// TwinCAT 3 PLC project TcMotionInterface_Test
// Title: TcMotionInterface_Test
// Company: TcInterfaces
// Author: R&B
// ProjectVersion: 1.0.0.0
// ProgramVersion: 3.1.4026.22
// CompilerDefines: ,VISU_USEPROPERTYINFO
// libraries:
//   Tc2_MC2, * (Beckhoff Automation GmbH)
//   Tc2_System, * (Beckhoff Automation GmbH)
//   Tc2_Utilities, * (Beckhoff Automation GmbH)
//   [TcMotionInterface], * (TcInterfaces)
//   VisuDialogs
// project tree:
//   / GlobalTextList.TcGTLO, PlcTask.TcTTO, PRG_TEST.TcPOU, Visualization Manager.TcVMO (not stored)
//   GVLs/ GVL.TcGVL
//   TESTs/ MotionTest.TcPOU (not stored), NcParameterTest.TcPOU (not stored), View_Test.TcVIS, XmlHandler_Test.TcPOU
// real-time tasks:
//   TASK PlcTask: cycle T#1ms, priority 6, ADS port 350
// motion (NC):
//   TASK NC-Task 1 SAF: cycle T#1ms, priority 4, ADS port 501
//   TASK NC-Task 1 SVB: cycle T#1ms, priority 8, ADS port 511
//   AXIS Axis1 (id 1)
//     MotionControl: Range=1, Time=1
//     OtherSettings: AllowMotionCmdToSlave=true
//     encoder EncType=16
//       EncPara: MaxCount=#x0000ffff
//     drive DrvType=13
//       Analog: TorqueSetpointScale=10, ScaleFactorActTorque=0.1
//       TimeComp: TaskDelayCycles=1
//     controller CtrType=1
//       CtrPara: PriorControlFactor=1
//         Observer: BandWidth=20
//   AXIS Axis2 (id 2)
//     OtherSettings: AllowMotionCmdToSlave=true
//     encoder EncType=16
//       EncPara: MaxCount=#x0000ffff
//     drive DrvType=13
//       Analog: TorqueSetpointScale=10, ScaleFactorActTorque=0.1
//       TimeComp: TaskDelayCycles=1
//     controller CtrType=1
//       CtrPara: PriorControlFactor=1
//         Observer: BandWidth=20
//   AXIS Axis3 (id 3)
//     OtherSettings: AllowMotionCmdToSlave=true
//     encoder EncType=16
//       EncPara: MaxCount=#x0000ffff
//     drive DrvType=13
//       Analog: TorqueSetpointScale=10, ScaleFactorActTorque=0.1
//       TimeComp: TaskDelayCycles=1
//     controller CtrType=1
//       CtrPara: PriorControlFactor=1
//         Observer: BandWidth=20
// variable links:
//   __THIS__ <-> TcMotionInterface_Test/TcMotionInterface_Test Instance
//     Inputs/FromPlc <-> PlcTask Outputs/GVL.axRef[0].PlcToNc
//     Inputs/FromPlc <-> PlcTask Outputs/GVL.axRef[1].PlcToNc
//     Inputs/FromPlc <-> PlcTask Outputs/GVL.axRef[2].PlcToNc
//     Outputs/ToPlc <-> PlcTask Inputs/GVL.axRef[0].NcToPlc
//     Outputs/ToPlc <-> PlcTask Inputs/GVL.axRef[1].NcToPlc
//     Outputs/ToPlc <-> PlcTask Inputs/GVL.axRef[2].NcToPlc
//   __THIS__ <-> MotionControllerLibrary/MotionControllerLibrary Instance
//     Inputs/FromPlc <-> PlcTask Outputs/GVL.axRef[0].PlcToNc
//     Inputs/FromPlc <-> PlcTask Outputs/GVL.axRef[1].PlcToNc
//     Inputs/FromPlc <-> PlcTask Outputs/GVL.axRef[2].PlcToNc
//     Outputs/ToPlc <-> PlcTask Inputs/GVL.axRef[0].NcToPlc
//     Outputs/ToPlc <-> PlcTask Inputs/GVL.axRef[1].NcToPlc
//     Outputs/ToPlc <-> PlcTask Inputs/GVL.axRef[2].NcToPlc
//   (this object) <-> TcMotionInterface_Test/TcMotionInterface_Test Instance
//     Inputs/FromPlc <-> PlcTask Outputs/GVL.axRef[0].PlcToNc
//     Inputs/FromPlc <-> PlcTask Outputs/GVL.axRef[1].PlcToNc
//     Inputs/FromPlc <-> PlcTask Outputs/GVL.axRef[2].PlcToNc
//     Outputs/ToPlc <-> PlcTask Inputs/GVL.axRef[0].NcToPlc
//     Outputs/ToPlc <-> PlcTask Inputs/GVL.axRef[1].NcToPlc
//     Outputs/ToPlc <-> PlcTask Inputs/GVL.axRef[2].NcToPlc

CONFIGURATION TcMotionInterface_Test
    RESOURCE PLC ON TwinCAT3
        TASK PlcTask(INTERVAL := T#1ms, PRIORITY := 6);
        PROGRAM PRG_TEST WITH PlcTask : PRG_TEST;
    END_RESOURCE
END_CONFIGURATION

// ---- GVLs/GVL.TcGVL
{attribute 'qualified_only'}
VAR_GLOBAL
	{attribute 'TcNcAxis' := '[0]:=Axis1; [1]:=Axis2; [2]:= Axis3'}
	axRef: ARRAY[0..2] OF AXIS_REF;
END_VAR

// ---- PRG_TEST.TcPOU
PROGRAM PRG_TEST
VAR
	Motion	: MotionTest;
	NC		: NcParameterTest;
	XML		: XmlHandler_Test;
END_VAR

Motion();
NC();
XML();

END_PROGRAM

// ---- TESTs/XmlHandler_Test.TcPOU
FUNCTION_BLOCK XmlHandler_Test
VAR
	XmlHandler: TcDriveParameterHandler;
	RouterMem: FB_GetRouterStatusInfo;
	Status: ST_TcRouterStatusInfo;
	file: STRING := '/home/Administrator/parm.xml';
	file2: STRING := '/home/Administrator/i550V5_4_Async50HzV1.xml';
	ax: AXIS_REF;
	write: BOOL;
	write2: BOOL;
	powerOn: BOOL;
	readState: BOOL;
	readAddr: BOOL;
	power: MC_Power;
	state: MC_ReadStatus;
	address: MC_ReadDriveAddress;
	reset: BOOL;
	starter: BOOL;
	startTime: ULINT;
	stopTime: ULINT;
	diffTime: ULINT;
	parametersWritten: UDINT;
	parametersWritten2: UDINT;
	canAms: STRING := '192.168.17.10.3.1';
	canNode: UINT := 14;
END_VAR

IF powerOn THEN
	power(Axis:= ax, 
		Enable:= TRUE, 
		Enable_Positive:= TRUE, 
		Enable_Negative:= TRUE
	);
END_IF

IF readState THEN
	state(Axis:= ax, Enable:= TRUE);
END_IF

IF readAddr THEN
	address(Axis:= ax, Execute:= TRUE);
END_IF

IF write and not write2 THEN
	IF NOT starter THEN
		startTime := F_GetSystemTime();
		starter := TRUE;
	END_IF
	
	IF XmlHandler.WriteEtcDriveParameter(FilePath:= file, NetId:= ax.DriveAddress.NetID, EtcAddress:= ax.DriveAddress.SlaveAddress, NumberOfParameterWritten=> parametersWritten) THEN
		stopTime := F_GetSystemTime();
		diffTime := (stopTime - startTime) / 10000; // ms
		starter := FALSE;
		write := FALSE;
	END_IF
	IF XmlHandler.Error THEN
		starter := FALSE;
		write := FALSE;
	END_IF
END_IF

IF write2 AND NOT write THEN
	IF NOT starter THEN
		startTime := F_GetSystemTime();
		starter := TRUE;
	END_IF
	
	IF XmlHandler.WriteCanOpenParameters(FilePath:= file2, NetId:= canAms, CanId:= canNode, NumberOfParameterWritten=> parametersWritten2) THEN
		stopTime := F_GetSystemTime();
		diffTime := (stopTime - startTime) / 10000; // ms
		starter := FALSE;
		write2 := FALSE;
	END_IF
	IF XmlHandler.Error THEN
		starter := FALSE;
		write2 := FALSE;
	END_IF
END_IF

IF reset THEN
	XmlHandler.ResetError();
	reset := FALSE;
END_IF

RouterMem(bExecute:= TRUE);
IF NOT RouterMem.bBusy THEN
	Status := RouterMem.info;
	RouterMem(bExecute:= FALSE);
END_IF

END_FUNCTION_BLOCK

// ---- GlobalTextList.TcGTLO
TEXTLIST GlobalTextList
  181 = '%d'
  185 = '%s'
  488 = 'Axis ID:'
  88 = 'Axis name to be saved in the JSON file.'
  699 = 'Axis name:'
  399 = 'Error: %s'
  637 = 'File name for the JSON to be saved to.\nWhite space it not allowed in the name.\n.json file extension is concated on the name.'
  377 = 'File name:'
  273 = 'File Path:'
  168 = 'Indicate if a parameter set have been loaded or read into the Visu.'
  169 = 'Load parameters'
  498 = 'Load the parameters from the JSON file'
  871 = 'NC Axis'
  455 = 'NC Axis parameters'
  689 = 'Parameter loaded:'
  309 = 'Path to where the JSON parameter file is loaded from and saved to.'
  68 = 'Read NC Axis'
  913 = 'Read the parameters from the NC Axis'
  731 = 'Reset any error that occured'
  105 = 'Reset error'
  645 = 'Save parameters'
  993 = 'Save the parameters to the JSON file'
  360 = 'Status: %s'
  599 = 'The axis ID in the Motion controller under the General tab.'
  774 = 'This Visu can be used for reading and writing to the NC Axis in the Motion controller.\nIt can also load and save the parameter to a JSON file on the OS.\nTo read and write the NC parameter, you need to provide a AxisID.\nTo load and save the parameter, you need to provide the file name and path to the file.\n'
  961 = 'Write NC Axis'
  216 = 'Write the parameters to the NC Axis'
END_TEXTLIST

// ---- TESTs/View_Test.TcVIS
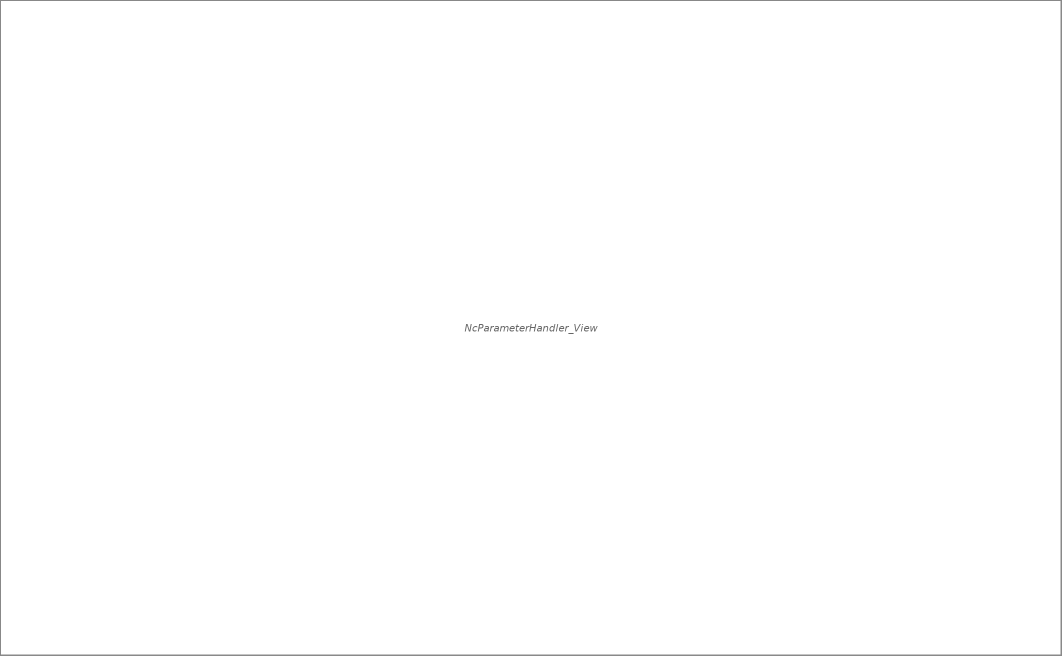
VISUALIZATION View_Test  // 1062x656
    TabControl (0,0 1062x656)
        shows NcParameterHandler_View(DataContent := PRG_TEST.NC.NcPHandler_VM)
        [0]: TabTitle=NC Axis
END_VISUALIZATION
